{attribute 'GeneratedUsingTerminal: AMP8000-0030-0103-0103'}
{attribute addProperty BoxType "AMP8000-0030-0103-0103"}
{attribute addProperty Id "Std_OutputBOOL1Std_Output_1BOOL1Std_Output_2BOOL1Std_Output_3BOOL1Std_Output_4BOOL1Std_Output_5BOOL1Std_Output_6BOOL1Std_Output_7BOOL1"}
{attribute addProperty CRC "3140699350"}
{attribute addProperty Size "8"}
TYPE FSOE_BB3344D6 :
STRUCT
	{attribute addProperty Name "Std_Output"}
	Std_Output : BOOL;
	{attribute addProperty Name "Std_Output_1"}
	Std_Output_1 : BOOL;
	{attribute addProperty Name "Std_Output_2"}
	Std_Output_2 : BOOL;
	{attribute addProperty Name "Std_Output_3"}
	Std_Output_3 : BOOL;
	{attribute addProperty Name "Std_Output_4"}
	Std_Output_4 : BOOL;
	{attribute addProperty Name "Std_Output_5"}
	Std_Output_5 : BOOL;
	{attribute addProperty Name "Std_Output_6"}
	Std_Output_6 : BOOL;
	{attribute addProperty Name "Std_Output_7"}
	Std_Output_7 : BOOL;
END_STRUCT
END_TYPE

(* stored: Version 1.2.0.0, ProductVersion 3.1.4024.9
   DUT FSOE_BB3344D6: Id {270c6751-1907-467c-86d3-89ace8c2e284} *)
